(* IEC 61131-3 sources: programs/VI-54/VI-54_20171205/VI-54_20171205/Stations/PLC_VI54/VI-54_171014/Class/DriveAxleErr, 1 file *)

(* ---- DriveAxleErr.st ---- *)
(*!
<Class
	Name               = "DriveAxleErr"
	Revision           = "6.1"
	RealtimeTask       = "false"
	CyclicTask         = "true"
	DefCyclictime      = "cCT"
	BackgroundTask     = "false"
	Sigmatek           = "false"
	OSInterface        = "false"
	HighPriority       = "false"
	Automatic          = "false"
	UpdateMode         = "Prescan"
	SharedCommandTable = "true"
	Objectsize         = "(570,480)">
	<Channels>
		<Server Name="DriveOnline" Visualized="false" Initialize="false" WriteProtected="true" Retentive="false"/>
		<Server Name="DrivesEnabled" Visualized="true" Initialize="false" WriteProtected="true" Retentive="false"/>
		<Server Name="DrivesOk" Visualized="true" Initialize="false" WriteProtected="false" Retentive="false"/>
		<Server Name="I_StatusNbr" Visualized="true" Initialize="false" WriteProtected="true" Retentive="false"/>
		<Server Name="ManagerEnabled" Visualized="true" Initialize="false" WriteProtected="true" Retentive="false"/>
	</Channels>
	<Network Name="DriveAxleErr">
		<!-- List of Components in this network -->
		<Components>
			<Object
				Name       = "_base"
				Class      = "_DriveErrorHandling"
				Position   = "(339,120)"
				Visualized = "true"
				Remotely   = "true">
				<Channels>
					<Server Name="GetErrorInfo"/>
					<Server Name="I_DERROR"/>
					<Server Name="I_STATUS"/>
					<Server Name="State"/>
					<Client Name="DriveAxis"/>
					<Client Name="ErrorCode"/>
				</Channels>
			</Object>
		</Components>
		<Comments>
		</Comments>
		<!-- List of Connections in this network -->
		<Connections>
			<Connection Source="_base.DriveAxis" Destination="this.DriveAxis" Vertices="(339,210),(38,210),"/>
			<Connection Source="_base.ErrorCode" Destination="this.ErrorCode" Vertices="(339,270),(38,270),"/>
			<Connection Source="this.State" Destination="_base.State" Vertices="(1067,210),(895,210),"/>
			<Connection Source="this.GetErrorInfo" Destination="_base.GetErrorInfo" Vertices="(1067,270),(895,270),"/>
			<Connection Source="this.I_STATUS" Destination="_base.I_STATUS" Vertices="(1067,330),(895,330),"/>
			<Connection Source="this.I_DERROR" Destination="_base.I_DERROR" Vertices="(1067,390),(895,390),"/>
		</Connections>
		<!-- Headerfiles -->
		<Options>
		</Options>
	</Network>
</Class>
*)
#pragma using _DriveErrorHandling

DriveAxleErr : CLASS
: _DriveErrorHandling
  //Servers:
	I_StatusNbr 	: SvrCh_DINT;
	DriveOnline 	: SvrCh_DINT;
	ManagerEnabled 	: SvrCh_DINT;
	DrivesOk 	: SvrCh_DINT;
	DrivesEnabled 	: SvrCh_DINT;
  //Clients:
  //Variables:
		cmdResetDrives 	: DINT;
		StateWord 	: DS402_State;
		DriveNoErrorOld 	: DINT;
		TestBits : BDINT
		[
		];

		TestNbr 	: DINT;
		DriveNoError 	: DINT;
		TmrReadStatus 	: UDINT;
		CntReadState 	: UDINT;
  //Functions:

	FUNCTION VIRTUAL GLOBAL CyWork
		VAR_INPUT
			EAX 	: UDINT;
		END_VAR
		VAR_OUTPUT
			state (EAX) 	: UDINT;
		END_VAR;

	FUNCTION GLOBAL ResetDrives;

	FUNCTION GLOBAL ReadDriveState
		VAR_OUTPUT
			State 	: DS402_State;
		END_VAR;

	FUNCTION GLOBAL ReadDriveOk
		VAR_OUTPUT
			State 	: DINT;
		END_VAR;

	FUNCTION GLOBAL ReadDriveEnabled
		VAR_OUTPUT
			State 	: DINT;
		END_VAR;

	FUNCTION GLOBAL ReadDriveOnline
		VAR_OUTPUT
			State 	: DINT;
		END_VAR;

	FUNCTION CheckBitNbr
		VAR_INPUT
			StateBits 	: BDINT;
		END_VAR
		VAR_OUTPUT
			BitNbr 	: DINT;
		END_VAR;

	FUNCTION VIRTUAL GLOBAL DrivesOk::Write
		VAR_INPUT
			input (EAX) 	: DINT;
		END_VAR
		VAR_OUTPUT
			result (EAX) 	: DINT;
		END_VAR;
  //Tables:
	FUNCTION @STD
		VAR_OUTPUT
			ret_code	: CONFSTATES;
		END_VAR;
	FUNCTION GLOBAL TAB @CT_;
END_CLASS;

FUNCTION VIRTUAL GLOBAL DriveAxleErr::CyWork
	VAR_INPUT
		EAX 	: UDINT;
	END_VAR
	VAR_OUTPUT
		state (EAX) 	: UDINT;
	END_VAR

  DriveOnline := (DriveAxis.IsOnline() = 1 & DriveAxis.Online.read() = 1);

  if DriveOnline = 1 then
    StateWord     := DriveAxis.StateWord.Read();
    ManagerEnabled  := (StateWord.SwitchedOn = 1);

    DrivesOk := I_STATUS = 0 & I_DERROR = 0; // check if we have a  axle error
    DriveNoError := DrivesOk;
    if DrivesOk = 1 then
      DrivesEnabled := (DriveAxis.AxOkay() = 1 & StateWord.OperationEnabled = 1); // no errors and enabled  !!
    else
      if cmdResetDrives = 1 then
        DriveAxis.ErrorQuitHandling(input:=1);
        // end of reset signal !!
        cmdResetDrives := 0;
      end_if;
      DrivesEnabled := 0;
    end_if;
  else
    DrivesOk      := 1;// not connected no error
    DrivesEnabled := 1;
    DriveNoError  := DrivesOk;
  end_if;

  // read as state !!
  if ops.tAbsolute - TmrReadStatus >= 100 then
    CntReadState += 1;
    GetErrorInfo.Write(1);
    TmrReadStatus := ops.tAbsolute;
  end_if;

  I_StatusNbr := CheckBitNbr(StateBits:= I_STATUS);

	state := READY;

END_FUNCTION

FUNCTION GLOBAL DriveAxleErr::ResetDrives

  cmdResetDrives := 1;  // give a reset command to de drives

END_FUNCTION

FUNCTION GLOBAL DriveAxleErr::ReadDriveState
	VAR_OUTPUT
		State 	: DS402_State;
	END_VAR

  State := StateWord;

END_FUNCTION

FUNCTION GLOBAL DriveAxleErr::ReadDriveOk
	VAR_OUTPUT
		State 	: DINT;
	END_VAR

  State := DrivesOk;

END_FUNCTION

FUNCTION GLOBAL DriveAxleErr::ReadDriveEnabled
	VAR_OUTPUT
		State 	: DINT;
	END_VAR

  State := DrivesEnabled;

END_FUNCTION

FUNCTION VIRTUAL GLOBAL DriveAxleErr::DrivesOk::Write
	VAR_INPUT
		input (EAX) 	: DINT;
	END_VAR
	VAR_OUTPUT
		result (EAX) 	: DINT;
	END_VAR

  if input = 1 then
    cmdResetDrives := input;
  end_if;

 	result := input;

END_FUNCTION

FUNCTION GLOBAL DriveAxleErr::ReadDriveOnline
	VAR_OUTPUT
		State 	: DINT;
	END_VAR

  State := DriveOnline;

END_FUNCTION

FUNCTION DriveAxleErr::CheckBitNbr
	VAR_INPUT
		StateBits 	: BDINT;
	END_VAR
	VAR_OUTPUT
		BitNbr 	: DINT;
	END_VAR
  VAR
  	MijnBit : BDINT;
  END_VAR

  BitNbr := 0;
  if StateBits <> 0 then
    repeat
    MijnBit := (StateBits AND 2#00000000000000000000000000000001);
    StateBits := (StateBits SHR 1);
    BitNbr += 1;
    until MijnBit = 1 | StateBits = 0 end_repeat;
  end_if;

END_FUNCTION
